SYSTEM DASDAass2 (* System Configuration *)
  (* Standard: 61499-1 *)
  (* Version 0.4, 2009-03-05, JHC, Holobloc Inc., Deleted Application. *)
  (* Version 0.3, 2003-12-05, JHC, Rockwell Automation, Renamed from NEWSYSTEM. *)
  (* Version 0.2, 2002-11-05, JHC, Rockwell Automation, Fixed missing (empty) FBD in Application. *)
  (* Version 0.1, 2002-01-17, JHC, Rockwell Automation, Minor cleanup *)
  (* Version 0.0, 2000-05-27, JHC, Rockwell Automation *)
  DEVICE HMI_LAYER : FRAME_DEVICE(BOUNDS := [0,0,200,200])
    RESOURCE HMI_1 : PANEL_RESOURCE(COLS := 1, ROWS := 0)
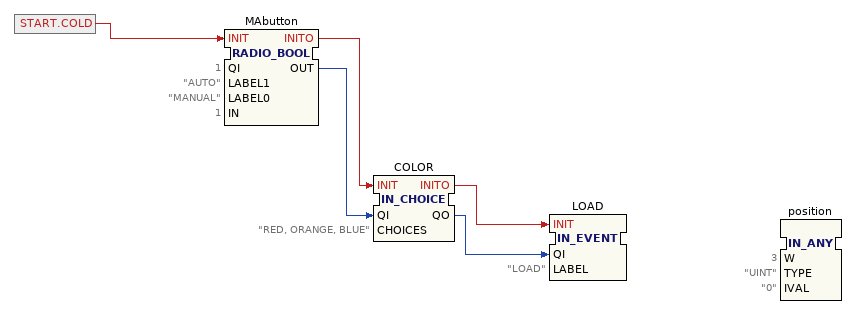
      FBS
        MAbutton : RADIO_BOOL(QI := 1, LABEL1 := "AUTO", LABEL0 := "MANUAL", IN := 1);
        LOAD : IN_EVENT(LABEL := "LOAD");
        COLOR : IN_CHOICE(CHOICES := "RED, ORANGE, BLUE");
        position : IN_ANY(W := 3, TYPE := "UINT", IVAL := "0");
      END_FBS
      EVENT_CONNECTIONS
        START.COLD TO MAbutton.INIT;
        COLOR.INITO TO LOAD.INIT;
        MAbutton.INITO TO COLOR.INIT;
      END_CONNECTIONS
      DATA_CONNECTIONS
        COLOR.QO TO LOAD.QI;
        MAbutton.OUT TO COLOR.QI;
      END_CONNECTIONS
    END_RESOURCE
  END_DEVICE
  DEVICE VIEW_LAYER : FRAME_DEVICE(BOUNDS := [250,0,900,900])
    RESOURCE VIEW_RES : VIEW_PANEL(DIA := 85, SIZE := [10,8], VERTICAL := 0)
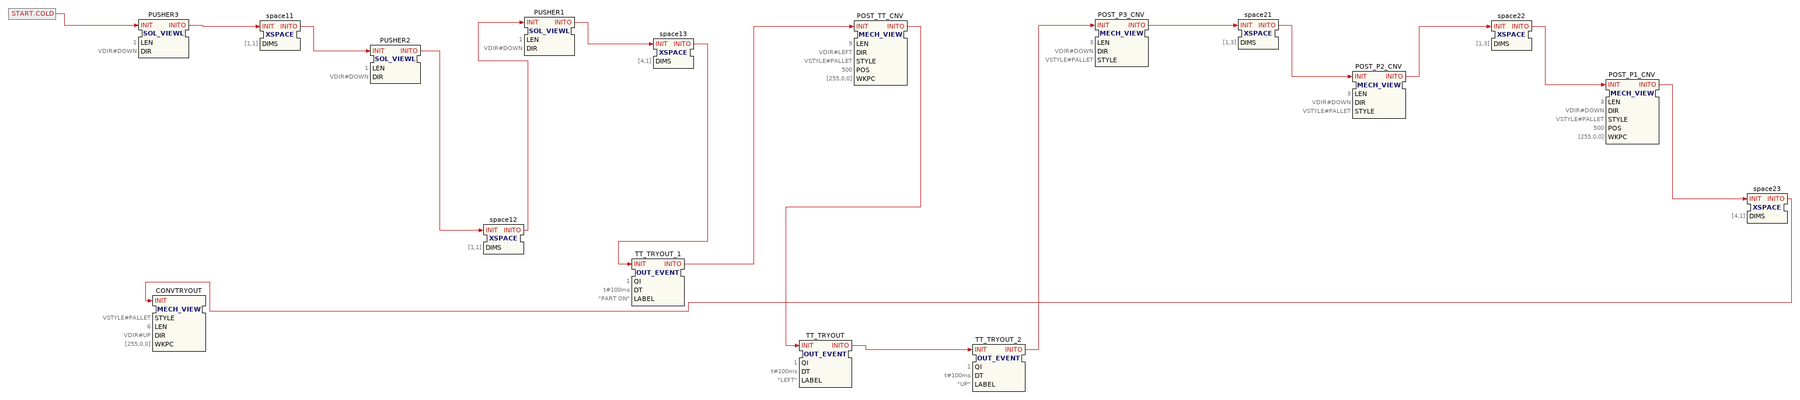
      FBS
        PUSHER3 : SOL_VIEWL(LEN := 1, DIR := VDIR#DOWN);
        space11 : XSPACE(DIMS := [1,1]);
        PUSHER2 : SOL_VIEWL(LEN := 1, DIR := VDIR#DOWN);
        space12 : XSPACE(DIMS := [1,1]);
        PUSHER1 : SOL_VIEWL(LEN := 1, DIR := VDIR#DOWN);
        space13 : XSPACE(DIMS := [4,1]);
        space21 : XSPACE(DIMS := [1,3]);
        space22 : XSPACE(DIMS := [1,3]);
        space23 : XSPACE(DIMS := [4,1]);
        POST_P1_CNV : MECH_VIEW(LEN := 3, DIR := VDIR#DOWN, STYLE := VSTYLE#PALLET, POS := 500, WKPC := [255,0,0]);
        POST_P2_CNV : MECH_VIEW(LEN := 3, DIR := VDIR#DOWN, STYLE := VSTYLE#PALLET);
        POST_P3_CNV : MECH_VIEW(LEN := 3, DIR := VDIR#DOWN, STYLE := VSTYLE#PALLET);
        POST_TT_CNV : MECH_VIEW(LEN := 9, DIR := VDIR#LEFT, STYLE := VSTYLE#PALLET, POS := 500, WKPC := [255,0,0]);
        TT_TRYOUT : OUT_EVENT(QI := 1, DT := t#100ms, LABEL := "LEFT");
        TT_TRYOUT_1 : OUT_EVENT(QI := 1, DT := t#100ms, LABEL := "PART ON");
        TT_TRYOUT_2 : OUT_EVENT(QI := 1, DT := t#100ms, LABEL := "UP");
        CONVTRYOUT : MECH_VIEW(STYLE := VSTYLE#PALLET, LEN := 6, DIR := VDIR#UP, WKPC := [255,0,0]);
      END_FBS
      EVENT_CONNECTIONS
        START.COLD TO PUSHER3.INIT;
        PUSHER3.INITO TO space11.INIT;
        space11.INITO TO PUSHER2.INIT;
        PUSHER2.INITO TO space12.INIT;
        space12.INITO TO PUSHER1.INIT;
        PUSHER1.INITO TO space13.INIT;
        space22.INITO TO POST_P1_CNV.INIT;
        POST_P1_CNV.INITO TO space23.INIT;
        space21.INITO TO POST_P2_CNV.INIT;
        POST_P2_CNV.INITO TO space22.INIT;
        POST_P3_CNV.INITO TO space21.INIT;
        POST_TT_CNV.INITO TO TT_TRYOUT.INIT;
        space13.INITO TO TT_TRYOUT_1.INIT;
        TT_TRYOUT_1.INITO TO POST_TT_CNV.INIT;
        TT_TRYOUT.INITO TO TT_TRYOUT_2.INIT;
        TT_TRYOUT_2.INITO TO POST_P3_CNV.INIT;
        space23.INITO TO CONVTRYOUT.INIT;
      END_CONNECTIONS
    END_RESOURCE
  END_DEVICE
  DEVICE MODEL_LAYER : FRAME_DEVICE
    RESOURCE MODEL_CLOCK : PANEL_RESOURCE
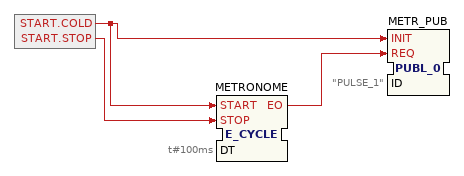
      FBS
        METRONOME : E_CYCLE(DT := t#100ms);
        METR_PUB : PUBL_0(ID := "PULSE_1");
      END_FBS
      EVENT_CONNECTIONS
        START.COLD TO METRONOME.START;
        START.COLD TO METR_PUB.INIT;
        METRONOME.EO TO METR_PUB.REQ;
        START.STOP TO METRONOME.STOP;
      END_CONNECTIONS
    END_RESOURCE
    RESOURCE CNV_1_MODEL : PANEL_RESOURCE
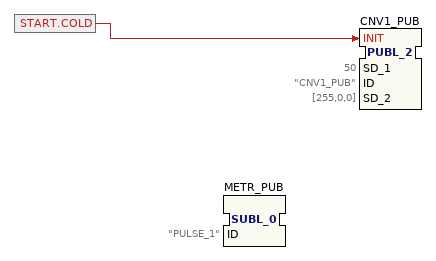
      FBS
        CNV1_PUB : PUBL_2(SD_1 := 50, ID := "CNV1_PUB", SD_2 := [255,0,0]);
        METR_PUB : SUBL_0(ID := "PULSE_1");
      END_FBS
      EVENT_CONNECTIONS
        START.COLD TO CNV1_PUB.INIT;
      END_CONNECTIONS
    END_RESOURCE
    RESOURCE TT_MODEL : PANEL_RESOURCE
    END_RESOURCE
    RESOURCE CNV_2_MODEL : PANEL_RESOURCE
    END_RESOURCE
    RESOURCE PUSHER1_MODEL : PANEL_RESOURCE
    END_RESOURCE
    RESOURCE PUSHER_2_MODEL : PANEL_RESOURCE
    END_RESOURCE
    RESOURCE PUSHER3_MODEL : PANEL_RESOURCE
    END_RESOURCE
  END_DEVICE
END_SYSTEM
